FUNCTION_BLOCK FB_CoE_EL3446
VAR_INPUT
	m_start: BOOL;
	nSlaveAddr	:UINT;
	b_SubIndex	:BYTE;
	uiVoltagePhaseSelector_CH1		: UINT;											//Voltage Phase Selector 1/2/3 for Channel 1
	uiVoltagePhaseSelector_CH2		: UINT;											//Voltage Phase Selector 1/2/3 for Channel 2
	uiVoltagePhaseSelector_CH3		: UINT;											//Voltage Phase Selector 1/2/3 for Channel 3
	uiVoltagePhaseSelector_CH4		: UINT;											//Voltage Phase Selector 1/2/3 for Channel 4
	uiVoltagePhaseSelector_CH5		: UINT;											//Voltage Phase Selector 1/2/3 for Channel 5
	uiVoltagePhaseSelector_CH6		: UINT;											//Voltage Phase Selector 1/2/3 for Channel 6 
END_VAR
VAR_OUTPUT
	m_Busy: BOOL;
	m_CoE_Write_done: BOOL;
	m_Error: bool;
	udint_GetAMSNetID_Error: UDINT;
	udint_WriteCoE_Error: UDINT;
END_VAR
VAR
	i_State	:UINT:=1;
	fb_GetAMSNetID	:FB_GetLocalAmsNetId;
  	fb_coe_write          : FB_EcCoESdoWrite; // Function Block for writing in CoE


	r_trig_Start: R_trig;
	i_errorCount: INT;
	i_AMSNetID_ReadOut_Succesfull: INT;
	str_AMSNetID: STRING(30);
 	nValue     : UdINT ; (* variable to be written to the CoE Object *)
 	
	i_CoE_Write_Succesfull: INT;
	udint_Value: UDINT;
	real_Value: REAL;

END_VAR


r_trig_Start(Clk := m_start);
b_SubIndex := LIMIT (1,b_SubIndex,8);
CASE i_State OF
	1: 		// wait for start
	IF r_trig_Start.Q THEN
		i_State := i_State+1;
		m_CoE_Write_done := FALSE;
		m_Busy := TRUE;
		m_Error := FALSE;
	END_IF

	2:		// read out ams net ID	
	fb_GetAMSNetID.bExecute := TRUE;
	i_State := i_State+1;
	
	3: 		// wait for read ot
	IF fb_GetAMSNetID.bBusy = FALSE AND NOT fb_GetAMSNetID.bError = TRUE THEN
		fb_GetAMSNetID.bExecute := FALSE;
		i_AMSNetID_ReadOut_Succesfull := i_AMSNetID_ReadOut_Succesfull+1;
		i_State := i_State+1;
	ELSIF fb_GetAMSNetID.bError = TRUE THEN
		fb_GetAMSNetID.bExecute := FALSE;
		i_State := 100;
	END_IF
	
	4: 		// read out AMS Net ID done, convert received data
	str_AMSNetID := concat(BYTE_TO_STRING(fb_GetAMSNetID.AddrBytes[0]),'.');
	str_AMSNetID := concat(str_AMSNetID,BYTE_TO_STRING(fb_GetAMSNetID.AddrBytes[1]));
	str_AMSNetID := concat(str_AMSNetID,'.');	
	str_AMSNetID := concat(str_AMSNetID,BYTE_TO_STRING(fb_GetAMSNetID.AddrBytes[2]));
	str_AMSNetID := concat(str_AMSNetID,'.');
	str_AMSNetID := concat(str_AMSNetID,BYTE_TO_STRING(fb_GetAMSNetID.AddrBytes[3]));
	str_AMSNetID := concat(str_AMSNetID,'.');
	str_AMSNetID := concat(str_AMSNetID,BYTE_TO_STRING(b_SubIndex));
	str_AMSNetID := concat(str_AMSNetID,'.1');
	
	i_State := 10;

	10: 	// write channel 1 phase Selector
	fb_coe_write.bExecute 	:= TRUE;
	fb_coe_write.nIndex		:= 16#8000;
	fb_coe_write.nSubIndex	:= 16#11; 
	udint_Value 			:= UINT_TO_UDINT(uiVoltagePhaseSelector_CH1);
	fb_coe_write.pSrcBuf	:= ADR(udint_Value);
	fb_coe_write.cbBufLen	:= SIZEOF(udint_Value);
	i_State := i_State+1;
	
	11: 	// wait for done or error
	IF NOT fb_coe_write.bBusy AND NOT fb_coe_write.bError THEN
		fb_coe_write.bExecute 	:= FALSE;
		i_CoE_Write_Succesfull := i_CoE_Write_Succesfull+1;
		i_State := i_State+1;
	ELSIF fb_coe_write.bError THEN
		fb_coe_write.bExecute 	:= FALSE;
		i_State := 100;
	END_IF

	12:		// wait 
	i_State := 20;
	
	20: 	// write channel 2 phase Selector
	fb_coe_write.bExecute 	:= TRUE;
	fb_coe_write.nIndex		:= 16#8010;
	fb_coe_write.nSubIndex	:= 16#11; 
	udint_Value 			:= UINT_TO_UDINT(uiVoltagePhaseSelector_CH2);
	fb_coe_write.pSrcBuf	:= ADR(udint_Value);
	fb_coe_write.cbBufLen	:= SIZEOF(udint_Value);
	i_State := i_State+1;
	
	21: 	// wait for done or error
	IF NOT fb_coe_write.bBusy AND NOT fb_coe_write.bError THEN
		fb_coe_write.bExecute 	:= FALSE;
		i_CoE_Write_Succesfull := i_CoE_Write_Succesfull+1;
		i_State := i_State+1;
	ELSIF fb_coe_write.bError THEN
		fb_coe_write.bExecute 	:= FALSE;
		i_State := 100;
	END_IF

	22:		// wait 
	i_State := 30;

	30: 	// write channel 3 phase Selector
	fb_coe_write.bExecute 	:= TRUE;
	fb_coe_write.nIndex		:= 16#8020;
	fb_coe_write.nSubIndex	:= 16#11; 
	udint_Value 			:= UINT_TO_UDINT(uiVoltagePhaseSelector_CH3);
	fb_coe_write.pSrcBuf	:= ADR(udint_Value);
	fb_coe_write.cbBufLen	:= SIZEOF(udint_Value);
	i_State := i_State+1;
	
	31: 	// wait for done or error
	IF NOT fb_coe_write.bBusy AND NOT fb_coe_write.bError THEN
		fb_coe_write.bExecute 	:= FALSE;
		i_CoE_Write_Succesfull := i_CoE_Write_Succesfull+1;
		i_State := i_State+1;
	ELSIF fb_coe_write.bError THEN
		fb_coe_write.bExecute 	:= FALSE;
		i_State := 100;
	END_IF

	32:		// wait 
	i_State := 40;
	
	40: 	// write channel 4 phase Selector
	fb_coe_write.bExecute 	:= TRUE;
	fb_coe_write.nIndex		:= 16#8030;
	fb_coe_write.nSubIndex	:= 16#11; 
	udint_Value 			:= UINT_TO_UDINT(uiVoltagePhaseSelector_CH4);
	fb_coe_write.pSrcBuf	:= ADR(udint_Value);
	fb_coe_write.cbBufLen	:= SIZEOF(udint_Value);
	i_State := i_State+1;
	
	41: 	// wait for done or error
	IF NOT fb_coe_write.bBusy AND NOT fb_coe_write.bError THEN
		fb_coe_write.bExecute 	:= FALSE;
		i_CoE_Write_Succesfull := i_CoE_Write_Succesfull+1;
		i_State := i_State+1;
	ELSIF fb_coe_write.bError THEN
		fb_coe_write.bExecute 	:= FALSE;
		i_State := 100;
	END_IF

	42:		// wait 
	i_State := 50;		

	50: 	// write channel 5 phase Selector
	fb_coe_write.bExecute 	:= TRUE;
	fb_coe_write.nIndex		:= 16#8040;
	fb_coe_write.nSubIndex	:= 16#11; 
	udint_Value 			:= UINT_TO_UDINT(uiVoltagePhaseSelector_CH5);
	fb_coe_write.pSrcBuf	:= ADR(udint_Value);
	fb_coe_write.cbBufLen	:= SIZEOF(udint_Value);
	i_State := i_State+1;
	
	51: 	// wait for done or error
	IF NOT fb_coe_write.bBusy AND NOT fb_coe_write.bError THEN
		fb_coe_write.bExecute 	:= FALSE;
		i_CoE_Write_Succesfull := i_CoE_Write_Succesfull+1;
		i_State := i_State+1;
	ELSIF fb_coe_write.bError THEN
		fb_coe_write.bExecute 	:= FALSE;
		i_State := 100;
	END_IF

	52:		// wait 
	i_State := 60;		

	60: 	// write channel 6 phase Selector
	fb_coe_write.bExecute 	:= TRUE;
	fb_coe_write.nIndex		:= 16#8050;
	fb_coe_write.nSubIndex	:= 16#11; 
	udint_Value 			:= UINT_TO_UDINT(uiVoltagePhaseSelector_CH6);
	fb_coe_write.pSrcBuf	:= ADR(udint_Value);
	fb_coe_write.cbBufLen	:= SIZEOF(udint_Value);
	i_State := i_State+1;
	
	61: 	// wait for done or error
	IF NOT fb_coe_write.bBusy AND NOT fb_coe_write.bError THEN
		fb_coe_write.bExecute 	:= FALSE;
		i_CoE_Write_Succesfull := i_CoE_Write_Succesfull+1;
		i_State := i_State+1;
	ELSIF fb_coe_write.bError THEN
		fb_coe_write.bExecute 	:= FALSE;
		i_State := 100;
	END_IF

	62:		// wait 
	m_CoE_Write_done := TRUE;
	m_Busy := FALSE;
	i_State := 1;		
	
	100: 	//error state
	i_errorCount := i_errorCount +1;
	udint_GetAMSNetID_Error := fb_GetAMSNetID.nErrId;
	udint_WriteCoE_Error := fb_coe_write.nErrId;
	m_Busy := FALSE;
	m_Error := true;
	i_State := 1;

END_CASE


fb_GetAMSNetID(
	bExecute:= , 
	tTimeOut:= T#2S, 
	bBusy=> , 
	bError=> , 
	nErrId=> , 
	AddrString=> , 
	AddrBytes=> );
	
fb_coe_write(
	sNetId:= str_AMSNetID, 
	nSlaveAddr:= nSlaveAddr, 
	nSubIndex:= , 
	nIndex:= , 
    pSrcBuf    := ,
    cbBufLen   := ,
	bExecute:= , 
	tTimeout:= T#2S , 
	bBusy=> , 
	bError=> , 
	nErrId=> );

END_FUNCTION_BLOCK

(* stored: Version 1.1.0.1, ProductVersion 3.1.4024.12
   POU FB_CoE_EL3446: Id {33fa00b6-3595-4c83-9d2d-7143fc5f9c84}, SpecialFunc None *)
